INTERFACE i_Traffic_Phase
VAR
	n_Phase_ID : INT;
END_VAR

END_INTERFACE

(* stored: Version 1.1.0.1
   Itf i_Traffic_Phase: Id {83da61c9-9c47-476d-8a97-e58859bf064a} *)
